// TIA Portal V17 export
// export: Created 2023-12-22T15:03:15.165634Z, ExportSetting WithDefaults, DisplayName Totally Integrated Automation Portal, DisplayVersion V17, DisplayName TIA Portal Openness, DisplayVersion V17, DisplayName TIA Portal Version Control Interface, DisplayVersion V17, DisplayName STEP 7 Professional, DisplayVersion V17, DisplayName STEP 7 Safety, DisplayVersion V17, DisplayName WinCC Advanced, DisplayVersion V17
DATA_BLOCK "KP_2_10_DB"   // DB520
VERSION : 0.1
// stored: AutoNumber false, DBAccessibleFromOPCUA true, DBAccessibleFromWebserver true, InstanceOfName KP_2_10, InstanceOfType FB
"KP_2_10"
   // VAR RETAIN
   //    limit { S7_SetPoint := 'True'} : Int := 2;
   //    load : Int;
   //    load_last : Int;
   //    KP { S7_SetPoint := 'True'} : Array[0..10] of "DRV_AUMA";
   //    load_ok { S7_SetPoint := 'True'} : Bool := TRUE;
   // END_VAR
BEGIN
   KP[0..10].Use.QF := FALSE;
   KP[0..10].Use.KM_Open := FALSE;
   KP[0..10].Use.KM_Close := FALSE;
   KP[0..10].Use.Open := TRUE;
   KP[0..10].Use.Close := TRUE;
   KP[0..10].Use.One_KM := FALSE;
   KP[0..10].Use.Air := FALSE;
   KP[0..10].Use.Cross := FALSE;
   KP[0..10].Use.CMD_Open := TRUE;
   KP[0..10].Use.CMD_Close := FALSE;
   KP[0..10].Use.Local_Keys := FALSE;
   KP[0..10].Use.CWF := FALSE;
   KP[0].Clock[0].SP := 10;
   KP[0].Clock[1..4].SP := 2;
   KP[1].Clock[0].SP := 10;
   KP[1].Clock[1..2].SP := 2;
   KP[1].Clock[3..4].SP := 99;
   KP[2].Clock[0].SP := 10;
   KP[2].Clock[1..2].SP := 2;
   KP[2].Clock[3..4].SP := 99;
   KP[3].Clock[0].SP := 10;
   KP[3].Clock[1..4].SP := 2;
   KP[4].Clock[0].SP := 10;
   KP[4].Clock[1..4].SP := 2;
   KP[5].Clock[0].SP := 10;
   KP[5].Clock[1..4].SP := 2;
   KP[6].Clock[0].SP := 10;
   KP[6].Clock[1..4].SP := 2;
   KP[7].Clock[0].SP := 10;
   KP[7].Clock[1..4].SP := 2;
   KP[8].Clock[0].SP := 10;
   KP[8].Clock[1..4].SP := 2;
   KP[9].Clock[0].SP := 10;
   KP[9].Clock[1..4].SP := 2;
   KP[10].Clock[0].SP := 10;
   KP[10].Clock[1..4].SP := 2;
   KP[0].CodeID := 0;
   KP[1].CodeID := 1;
   KP[2].CodeID := 2;
   KP[3..10].CodeID := 0;
   KP[0..10].Speed := 16#00;
END_DATA_BLOCK
